# B&R Automation Studio project AS_Target_Simulink_Test
Automation Studio 4.5.2.102; This project is for testing the As Target for simulink (Third-Party Program).

## Configuration Config1

CPU PC_any, AutomationRuntime D4.52, Build 4.1.2, Vc V4.52.0

### Hardware
```
PC : PC_any v1.1.0.0 (OrderNumber=PC)
  ConfigurationID = AS_Target_Simulink_Test_Config1
  SystemTick = 1000
  Cyclic1Duration = 10000
  Cyclic1Tolerance = 10000
  ActivateOpcUa = 1
  OpcUaPort = 4841
  OpcUa_AuthenticationSecurityPolicy_EnableNone = 1
  OpcUaInformationModels_PV_Version = 1
```

## Logical view

Binary libraries used (declarations not repeated): operator, runtime, astime, AsIecCon, brsystem, sys_lib, AsArLog, AsTCP

### Global.typ - Global data types
```iecst
TYPE
	myOutputType : 	STRUCT
		out_Real : REAL;
		out_Int : ARRAY[0..2]OF INT;
		out_Bool : BOOL;
	END_STRUCT;
	myInputType : 	STRUCT
		in_Real : REAL;
		in_Int : ARRAY[0..2]OF INT;
		New_Member : BOOL;
	END_STRUCT;
END_TYPE
```

### Global.var - Global variables
```iecst
VAR
	start : BOOL := FALSE;
	ref : LREAL := 0; (*Reference input*)
	reset : BOOL := FALSE;
	x : ARRAY[0..3] OF LREAL := [4(0)]; (*Inverted pendulum state x*)
	y : ARRAY[0..1] OF LREAL := [2(0)]; (*Inverted pendulum output y*)
	F : LREAL := 0; (*Car force*)
END_VAR
```

### Package Logical/Libraries - Global libraries

### Library Logical/Libraries/pctr_fun (ANSIC, version 1.00.0)

#### lib_properties.txt
```
For manual assignment to hardware configuration please
add the following additional include directories:

\Logical\MATLAB_includes\R2019b\

And the following additional build options:

-lm -D MODEL=pend_ctrl_fun -D NUMST=1 -D NCSTATES=0 -D HAVESTDIO -D MODEL_HAS_DYNAMICALLY_LOADED_SFCNS=0 -D CLASSIC_INTERFACE=0 -D ALLOCATIONFCN=0 -D TID01EQ=0 -D TERMFCN=1 -D ONESTEPFCN=1 -D MAT_FILE=0 -D MULTI_INSTANCE_CODE=1 -D INTEGER_CODE=0 -D MT=0
```

#### pctrFub.c
```c
/********************************************************************
 * COPYRIGHT -- Bernecker + Rainer Industrie-Elektronik Ges.m.b.H.
 ********************************************************************
 * Program: pend_ctrl_fun
 * File: pctrFub.c
 * Author: Bernecker + Rainer Industrie Elektronik Ges.m.b.H.
 * Created: Wed Mar 17 14:21:47 2010
 ********************************************************************
 * Implementation of program pend_ctrl_fun
 ********************************************************************
 * Generated with B&R Automation Studio Target for Simulink  V6.1.0
 * (ERT based)
 ********************************************************************/

#include <bur/plctypes.h>
#include "pend_ctrl_fun.h"
#include "rtwtypes.h"

/* Defines */
#define SS_TERMINATE 4
#define SS_OUTPUT 3
#define SS_INITIALIZE 2

/*  Data Types */

/**************************** GLOBAL DATA *************************************/
/*  Definitions */

/*  Declarations  */

/***************************** FILE SCOPE DATA ********************************/

/*************************** FUNCTIONS ****************************************/
#ifdef __cplusplus

unsigned long bur_heap_size = 6553500;

#endif

/*LEGACYMODE_VARIABLES*/
void pctrFub(struct pctrFub* inst)
{
  tag_RTM_pend_ctrl_fun* const pend_ctrl_fun_M = &(inst)->bur_pend_ctrl_fun;
	inst->bur_pend_ctrl_fun.blockIO = &(inst)->bur_BlockIO_pend_ctrl_fun;
	inst->bur_pend_ctrl_fun.dwork = &(inst)->bur_D_Work_pend_ctrl_fun;

  switch (inst->ssMethodType)
  {
   case SS_INITIALIZE:
    /* call model initialize function */
    pend_ctrl_fun_initialize(pend_ctrl_fun_M, inst);
    break;

   case SS_OUTPUT:
    /* call model step function */
    pend_ctrl_fun_step(pend_ctrl_fun_M, inst);

    break;

   case SS_TERMINATE:
    /* call model terminate function */
    pend_ctrl_fun_terminate(pend_ctrl_fun_M, inst);
    break;
  }
}

/*****************************************************************************
   Function block sample time: 0.01s
 *****************************************************************************/

/*****************************************************************************
   B&R Automation Studio Target for Simulink Version: A6.1.0 (06-Nov-2019)
 *****************************************************************************/

/*======================== TOOL VERSION INFORMATION ==========================*
 * MATLAB 9.7 (R2019b)18-Jul-2019                                             *
 * Simulink 10.0 (R2019b)18-Jul-2019                                          *
 * Simulink Coder 9.2 (R2019b)18-Jul-2019                                     *
 * Embedded Coder 7.3 (R2019b)18-Jul-2019                                     *
 * Stateflow 10.1 (R2019b)18-Jul-2019                                         *
 * Fixed-Point Designer 6.4 (R2019b)18-Jul-2019                               *
 *============================================================================*/

/*======================= LICENSE IN USE INFORMATION =========================*
 * control_toolbox                                                            *
 * image_toolbox                                                              *
 * matlab                                                                     *
 * matlab_coder                                                               *
 * opc_toolbox                                                                *
 * real-time_workshop                                                         *
 * rtw_embedded_coder                                                         *
 * simulink                                                                   *
 *============================================================================*/
```

#### pctr_fun.fun
```iecst
FUNCTION_BLOCK pctrFub
	VAR_INPUT
		ssMethodType : SINT;
		ref : LREAL; (*Reference input*)
		x : ARRAY[0..3] OF LREAL; (*Inverted pendulum state x*)
		y : ARRAY[0..1] OF LREAL; (*Inverted pendulum output y*)
	END_VAR
	VAR_OUTPUT
		err_code : UINT; (*Controller error code*)
		F : LREAL; (*Car force*)
	END_VAR
	VAR
		bur_BlockIO_pend_ctrl_fun : BlockIO_pend_ctrl_fun;
		bur_D_Work_pend_ctrl_fun : D_Work_pend_ctrl_fun;
		bur_pend_ctrl_fun : tag_RTM_pend_ctrl_fun;
	END_VAR
END_FUNCTION_BLOCK
```

#### pctr_fun.typ
```iecst
TYPE
	BlockIO_pend_ctrl_fun :  STRUCT
		Input :  LREAL;
		Input_b :  ARRAY[0..3] OF LREAL;
		Input1 :  ARRAY[0..1] OF LREAL;
		u :  LREAL;
		err_code :  UINT;
	END_STRUCT;

	D_Work_pend_ctrl_fun :  STRUCT
		local_err_code :  UINT;
	END_STRUCT;

	tag_RTM_pend_ctrl_fun :  STRUCT
		errorStatus :  REFERENCE TO USINT;
		blockIO :  REFERENCE TO BlockIO_pend_ctrl_fun;
		dwork :  REFERENCE TO D_Work_pend_ctrl_fun;
	END_STRUCT;

	RT_MODEL_pend_ctrl_fun :tag_RTM_pend_ctrl_fun;	(*  *)

END_TYPE
```

#### pend_ctrl_fun.c
```c
/********************************************************************
 * COPYRIGHT -- Bernecker + Rainer Industrie-Elektronik Ges.m.b.H.
 ********************************************************************
 * Program: pend_ctrl_fun
 * File: pend_ctrl_fun.c
 * Author: Bernecker + Rainer Industrie Elektronik Ges.m.b.H.
 * Created: Wed Mar 17 14:21:47 2010
 ********************************************************************
 * Implementation of program pend_ctrl_fun
 ********************************************************************
 * Generated with B&R Automation Studio Target for Simulink  V6.1.0
 * (ERT based)
 ********************************************************************/

#include "pend_ctrl_fun.h"
#include "pend_ctrl_fun_private.h"

/*  Defines */

/*  Data Types */

/**************************** GLOBAL DATA *************************************/
/*  Definitions */

/*  Declarations  */

/***************************** FILE SCOPE DATA ********************************/

/*************************** FUNCTIONS ****************************************/

/* Model step function */
void pend_ctrl_fun_step(RT_MODEL_pend_ctrl_fun *const pend_ctrl_fun_M, struct pctrFub* inst)
{
  struct BlockIO_pend_ctrl_fun *pend_ctrl_fun_B = ((struct BlockIO_pend_ctrl_fun *)
    pend_ctrl_fun_M->blockIO);
  struct D_Work_pend_ctrl_fun *pend_ctrl_fun_DWork = ((struct D_Work_pend_ctrl_fun *)
    pend_ctrl_fun_M->dwork);
  real_T ref;
  uint16_T err_code;
  boolean_T varargin_1_idx_0;

  /* S-Function (bur_in): '<S1>/Input' */
  pend_ctrl_fun_B->Input = inst->ref;

  /* S-Function (bur_in): '<S4>/Input' */
  pend_ctrl_fun_B->Input_b[0] = inst->x[0];
  pend_ctrl_fun_B->Input_b[1] = inst->x[1];
  pend_ctrl_fun_B->Input_b[2] = inst->x[2];
  pend_ctrl_fun_B->Input_b[3] = inst->x[3];

  /* MATLAB Function: '<Root>/State feedback controller  with error handling' incorporates:
   *  Constant: '<Root>/ref_limit'
   *  Constant: '<Root>/u_limit'
   */
  ref = pend_ctrl_fun_B->Input;

  /* MATLAB Function 'State feedback controller  with error handling': '<S3>:1' */
  /* '<S3>:1:25' */
  err_code = pend_ctrl_fun_DWork->local_err_code;
  varargin_1_idx_0 = (fabs(pend_ctrl_fun_B->Input_b[0]) > 100.0);
  varargin_1_idx_0 = (((int32_T)varargin_1_idx_0 < (fabs
    (pend_ctrl_fun_B->Input_b[1]) > 100.0)) || varargin_1_idx_0);
  varargin_1_idx_0 = (((int32_T)varargin_1_idx_0 < (fabs
    (pend_ctrl_fun_B->Input_b[2]) > 100.0)) || varargin_1_idx_0);
  varargin_1_idx_0 = (((int32_T)varargin_1_idx_0 < (fabs
    (pend_ctrl_fun_B->Input_b[3]) > 100.0)) || varargin_1_idx_0);
  if (varargin_1_idx_0) {
    /* '<S3>:1:27' */
    /* '<S3>:1:28' */
    err_code = 50001U;

    /* '<S3>:1:29' */
    ref = 0.0;
  } else {
    if (pend_ctrl_fun_B->Input > 1.5) {
      /* '<S3>:1:31' */
      /* '<S3>:1:32' */
      err_code = 50013U;

      /* '<S3>:1:33' */
      ref = 1.5;
    } else {
      if (pend_ctrl_fun_B->Input < -1.5) {
        /* '<S3>:1:34' */
        /* '<S3>:1:35' */
        err_code = 50014U;

        /* '<S3>:1:36' */
        ref = -1.5;
      }
    }

    /* '<S3>:1:38' */
    ref = (((2987.4616903679125 * pend_ctrl_fun_B->Input_b[0] +
             3740.1178916812455 * pend_ctrl_fun_B->Input_b[1]) +
            32774.860875805127 * pend_ctrl_fun_B->Input_b[2]) +
           7399.4348019785593 * pend_ctrl_fun_B->Input_b[3]) +
      -2987.4616903679112 * ref;
    if (ref > 10000.0) {
      /* '<S3>:1:39' */
      /* '<S3>:1:40' */
      ref = 10000.0;

      /* '<S3>:1:41' */
      err_code = 50011U;
    } else {
      if (ref < -10000.0) {
        /* '<S3>:1:42' */
        /* '<S3>:1:43' */
        ref = -10000.0;

        /* '<S3>:1:44' */
        err_code = 50012U;
      }
    }
  }

  /* '<S3>:1:47' */
  pend_ctrl_fun_DWork->local_err_code = err_code;
  pend_ctrl_fun_B->u = ref;
  pend_ctrl_fun_B->err_code = err_code;

  /* End of MATLAB Function: '<Root>/State feedback controller  with error handling' */

  /* S-Function (bur_out): '<Root>/Output' */
  inst->err_code = pend_ctrl_fun_B->err_code;

  /* S-Function (bur_in): '<S4>/Input1' */
  pend_ctrl_fun_B->Input1[0] = inst->y[0];
  pend_ctrl_fun_B->Input1[1] = inst->y[1];

  /* S-Function (bur_out): '<S4>/Output' */
  inst->F = pend_ctrl_fun_B->u;
}

/* Model initialize function */
void pend_ctrl_fun_initialize(RT_MODEL_pend_ctrl_fun *const pend_ctrl_fun_M, struct pctrFub* inst)
{
  /* (no initialization code required) */
  UNUSED_PARAMETER(pend_ctrl_fun_M);
}

/* Model terminate function */
void pend_ctrl_fun_terminate(RT_MODEL_pend_ctrl_fun *const pend_ctrl_fun_M, struct pctrFub* inst)
{
  /* (no terminate code required) */
  UNUSED_PARAMETER(pend_ctrl_fun_M);
}

/*======================== TOOL VERSION INFORMATION ==========================*
 * MATLAB 9.7 (R2019b)18-Jul-2019                                             *
 * Simulink 10.0 (R2019b)18-Jul-2019                                          *
 * Simulink Coder 9.2 (R2019b)18-Jul-2019                                     *
 * Embedded Coder 7.3 (R2019b)18-Jul-2019                                     *
 * Stateflow 10.1 (R2019b)18-Jul-2019                                         *
 * Fixed-Point Designer 6.4 (R2019b)18-Jul-2019                               *
 *============================================================================*/

/*======================= LICENSE IN USE INFORMATION =========================*
 * control_toolbox                                                            *
 * image_toolbox                                                              *
 * matlab                                                                     *
 * matlab_coder                                                               *
 * opc_toolbox                                                                *
 * real-time_workshop                                                         *
 * rtw_embedded_coder                                                         *
 * simulink                                                                   *
 *============================================================================*/
```

#### pend_ctrl_fun.h
```c
/********************************************************************
 * COPYRIGHT -- Bernecker + Rainer Industrie-Elektronik Ges.m.b.H.
 ********************************************************************
 * Program: pend_ctrl_fun
 * File: pend_ctrl_fun.h
 * Author: Bernecker + Rainer Industrie Elektronik Ges.m.b.H.
 * Created: Wed Mar 17 14:21:47 2010
 ********************************************************************
 * Header for program pend_ctrl_fun
 ********************************************************************
 * Generated with B&R Automation Studio Target for Simulink  V6.1.0
 * (ERT based)
 ********************************************************************/

#ifndef RTW_HEADER_pend_ctrl_fun_h_
#define RTW_HEADER_pend_ctrl_fun_h_
#include <math.h>
#ifndef pend_ctrl_fun_COMMON_INCLUDES_
# define pend_ctrl_fun_COMMON_INCLUDES_
#include "rtwtypes.h"
#endif                                 /* pend_ctrl_fun_COMMON_INCLUDES_ */

#include "pend_ctrl_fun_types.h"
#include "pctr_fun.h"
/* Beginning of Dynamic TypeDefs: */
/* End of Dynamic TypeDefs: */
#ifndef MIN
#define MIN(a,b)	((a) < (b) ? (a) : (b))
#endif

#ifndef MAX
#define MAX(a,b)	((a) > (b) ? (a) : (b))
#endif

#ifndef AST_ROUND
#define AST_ROUND(x) ((x)>=0?(long long)((x)+0.5):(long long)((x)-0.5))
#endif

#include "rt_defines.h"

/* Macros for accessing real-time model data structure */
#ifndef rtmGetBlockIO
# define rtmGetBlockIO(rtm)            ((rtm)->blockIO)
#endif

#ifndef rtmSetBlockIO
# define rtmSetBlockIO(rtm, val)       ((rtm)->blockIO = (val))
#endif

#ifndef rtmGetRootDWork
# define rtmGetRootDWork(rtm)          ((rtm)->dwork)
#endif

#ifndef rtmSetRootDWork
# define rtmSetRootDWork(rtm, val)     ((rtm)->dwork = (val))
#endif

#ifndef rtmGetErrorStatus
# define rtmGetErrorStatus(rtm)        ((rtm)->errorStatus)
#endif

#ifndef rtmSetErrorStatus
# define rtmSetErrorStatus(rtm, val)   ((rtm)->errorStatus = (val))
#endif

#ifndef MIN
#define MIN(a,b)                       ((a) < (b) ? (a) : (b))
#endif

#ifndef MAX
#define MAX(a,b)                       ((a) > (b) ? (a) : (b))
#endif

/* Block signals (default storage) */

/* Block states (default storage) for system '<Root>' */

/* Real-time Model Data Structure */

/* Model entry point functions */
extern void pend_ctrl_fun_initialize(RT_MODEL_pend_ctrl_fun *const
  pend_ctrl_fun_M, struct pctrFub* inst);
extern void pend_ctrl_fun_step(RT_MODEL_pend_ctrl_fun *const pend_ctrl_fun_M, struct pctrFub* inst);
extern void pend_ctrl_fun_terminate(RT_MODEL_pend_ctrl_fun *const
  pend_ctrl_fun_M, struct pctrFub* inst);

/*-
 * The generated code includes comments that allow you to trace directly
 * back to the appropriate location in the model.  The basic format
 * is <system>/block_name, where system is the system number (uniquely
 * assigned by Simulink) and block_name is the name of the block.
 *
 * Use the MATLAB hilite_system command to trace the generated code back
 * to the model.  For example,
 *
 * hilite_system('<S3>')    - opens system 3
 * hilite_system('<S3>/Kp') - opens and selects block Kp which resides in S3
 *
 * Here is the system hierarchy for this model
 *
 * '<Root>' : 'pend_ctrl_fun'
 * '<S1>'   : 'pend_ctrl_fun/B&R reference input'
 * '<S2>'   : 'pend_ctrl_fun/Inverted Pendulum (Simulation // IOs)'
 * '<S3>'   : 'pend_ctrl_fun/State feedback controller  with error handling'
 * '<S4>'   : 'pend_ctrl_fun/Inverted Pendulum (Simulation // IOs)/inverted_pendulum_IOs'
 */
#endif                                 /* RTW_HEADER_pend_ctrl_fun_h_ */
```

#### pend_ctrl_fun_private.h
```c
/********************************************************************
 * COPYRIGHT -- Bernecker + Rainer Industrie-Elektronik Ges.m.b.H.
 ********************************************************************
 * Program: pend_ctrl_fun
 * File: pend_ctrl_fun_private.h
 * Author: Bernecker + Rainer Industrie Elektronik Ges.m.b.H.
 * Created: Wed Mar 17 14:21:47 2010
 ********************************************************************
 * Header for program pend_ctrl_fun
 ********************************************************************
 * Generated with B&R Automation Studio Target for Simulink  V6.1.0
 * (ERT based)
 ********************************************************************/

#ifndef RTW_HEADER_pend_ctrl_fun_private_h_
#define RTW_HEADER_pend_ctrl_fun_private_h_
#include "rtwtypes.h"
#include <bur/plctypes.h>
#ifndef MIN
#define MIN(a,b)                       ((a) < (b) ? (a) : (b))
#endif

#ifndef MAX
#define MAX(a,b)                       ((a) > (b) ? (a) : (b))
#endif
#endif                                 /* RTW_HEADER_pend_ctrl_fun_private_h_ */
```

#### pend_ctrl_fun_types.h
```c
/********************************************************************
 * COPYRIGHT -- Bernecker + Rainer Industrie-Elektronik Ges.m.b.H.
 ********************************************************************
 * Program: pend_ctrl_fun
 * File: pend_ctrl_fun_types.h
 * Author: Bernecker + Rainer Industrie Elektronik Ges.m.b.H.
 * Created: Wed Mar 17 14:21:47 2010
 ********************************************************************
 * Header for program pend_ctrl_fun
 ********************************************************************
 * Generated with B&R Automation Studio Target for Simulink  V6.1.0
 * (ERT based)
 ********************************************************************/

#ifndef RTW_HEADER_pend_ctrl_fun_types_h_
#define RTW_HEADER_pend_ctrl_fun_types_h_
#ifndef MIN
#define MIN(a,b)                       ((a) < (b) ? (a) : (b))
#endif

#ifndef MAX
#define MAX(a,b)                       ((a) > (b) ? (a) : (b))
#endif

/* Forward declaration for rtModel */

#endif                                 /* RTW_HEADER_pend_ctrl_fun_types_h_ */
```

#### rt_defines.h
```c
/********************************************************************
 * COPYRIGHT -- Bernecker + Rainer Industrie-Elektronik Ges.m.b.H.
 ********************************************************************
 * Program: pend_ctrl_fun
 * File: rt_defines.h
 * Author: Bernecker + Rainer Industrie Elektronik Ges.m.b.H.
 * Created: Wed Mar 17 14:21:47 2010
 ********************************************************************
 * Header for program pend_ctrl_fun
 ********************************************************************
 * Generated with B&R Automation Studio Target for Simulink  V6.1.0
 * (ERT based)
 ********************************************************************/

#ifndef RTW_HEADER_rt_defines_h_
#define RTW_HEADER_rt_defines_h_
#ifndef MIN
#define MIN(a,b)                       ((a) < (b) ? (a) : (b))
#endif

#ifndef MAX
#define MAX(a,b)                       ((a) > (b) ? (a) : (b))
#endif

/*===========*
 * Constants *
 *===========*/
#define RT_PI                          3.14159265358979323846
#define RT_PIF                         3.1415927F
#define RT_LN_10                       2.30258509299404568402
#define RT_LN_10F                      2.3025851F
#define RT_LOG10E                      0.43429448190325182765
#define RT_LOG10EF                     0.43429449F
#define RT_E                           2.7182818284590452354
#define RT_EF                          2.7182817F

/*
 * UNUSED_PARAMETER(x)
 *   Used to specify that a function parameter (argument) is required but not
 *   accessed by the function body.
 */
#ifndef UNUSED_PARAMETER
# if defined(__LCC__)
#   define UNUSED_PARAMETER(x)                                   /* do nothing */
# else

/*
 * This is the semi-ANSI standard way of indicating that an
 * unused function parameter is required.
 */
#   define UNUSED_PARAMETER(x)         (void) (x)
# endif
#endif
#endif                                 /* RTW_HEADER_rt_defines_h_ */
```

#### rtwtypes.h
```c
/********************************************************************
 * COPYRIGHT -- Bernecker + Rainer Industrie-Elektronik Ges.m.b.H.
 ********************************************************************
 * Program: pend_ctrl_fun
 * File: rtwtypes.h
 * Author: Bernecker + Rainer Industrie Elektronik Ges.m.b.H.
 * Created: Wed Mar 17 14:21:47 2010
 ********************************************************************
 * Header for program pend_ctrl_fun
 ********************************************************************
 * Generated with B&R Automation Studio Target for Simulink  V6.1.0
 * (ERT based)
 ********************************************************************/

#ifndef RTWTYPES_H
#define RTWTYPES_H

/* Logical type definitions */
#if (!defined(__cplusplus))
#  ifndef false
#   define false                       (0U)
#  endif

#  ifndef true
#   define true                        (1U)
#  endif
#endif

/*=======================================================================*
 * Target hardware information
 *   Device type: Intel->x86/Pentium
 *   Number of bits:     char:   8    short:   16    long:  32
 *                       long:  32
 *                       native word size:  32
 *   Byte ordering: LittleEndian
 *   Signed integer division rounds to: Zero
 *   Shift right on a signed integer as arithmetic shift: on
 *=======================================================================*/

/*=======================================================================*
 * Fixed width word size data types:                                     *
 *   int8_T, int16_T, int32_T     - signed 8, 16, or 32 bit integers     *
 *   uint8_T, uint16_T, uint32_T  - unsigned 8, 16, or 32 bit integers   *
 *   real32_T, real64_T           - 32 and 64 bit floating point numbers *
 *=======================================================================*/
typedef signed char int8_T;
typedef unsigned char uint8_T;
typedef short int16_T;
typedef unsigned short uint16_T;
typedef long int32_T;
typedef unsigned long uint32_T;
typedef float real32_T;
typedef double real64_T;

/*===========================================================================*
 * Generic type definitions: boolean_T, char_T, byte_T, int_T, uint_T,       *
 *                           real_T, time_T, ulong_T.                        *
 *===========================================================================*/
typedef double real_T;
typedef double time_T;
typedef unsigned char boolean_T;
typedef long int_T;
typedef unsigned long uint_T;
typedef unsigned long ulong_T;
typedef char char_T;
typedef unsigned char uchar_T;
typedef char_T byte_T;

/*=======================================================================*
 * Min and Max:                                                          *
 *   int8_T, int16_T, int32_T     - signed 8, 16, or 32 bit integers     *
 *   uint8_T, uint16_T, uint32_T  - unsigned 8, 16, or 32 bit integers   *
 *=======================================================================*/
#define MAX_int8_T                     ((int8_T)(127))
#define MIN_int8_T                     ((int8_T)(-128))
#define MAX_uint8_T                    ((uint8_T)(255U))
#define MAX_int16_T                    ((int16_T)(32767))
#define MIN_int16_T                    ((int16_T)(-32768))
#define MAX_uint16_T                   ((uint16_T)(65535U))
#define MAX_int32_T                    ((int32_T)(2147483647))
#define MIN_int32_T                    ((int32_T)(-2147483647-1))
#define MAX_uint32_T                   ((uint32_T)(0xFFFFFFFFU))

/* Block D-Work pointer type */
typedef void * pointer_T;

#endif                                 /* RTWTYPES_H */

#ifndef MIN
#define MIN(a,b)                       ((a) < (b) ? (a) : (b))
#endif

#ifndef MAX
#define MAX(a,b)                       ((a) > (b) ? (a) : (b))
#endif
```

### Package Logical/MATLAB_includes - Default includes for B&R Automation Studio Target for Simulink

### MatlabDataArray.hpp
```cpp
/* Copyright 2016-2017 The MathWorks, Inc. */

#ifndef MATLAB_DATA_ARRAY_HPP
#define MATLAB_DATA_ARRAY_HPP

#include "MatlabDataArray/Exception.hpp"
#include "MatlabDataArray/matlab_data_array_defs.hpp"
#include "MatlabDataArray/matlab_extdata_defs.hpp"
#include "MatlabDataArray/ArrayDimensions.hpp"
#include "MatlabDataArray/ArrayType.hpp"
#include "MatlabDataArray/GetReturnType.hpp"
#include "MatlabDataArray/Range.hpp"
#include "MatlabDataArray/String.hpp"
#include "MatlabDataArray/Enumeration.hpp"
#include "MatlabDataArray/Struct.hpp"
#include "MatlabDataArray/Reference.hpp"
#include "MatlabDataArray/ArrayElementRef.hpp"
#include "MatlabDataArray/ArrayElementTypedRef.hpp"
#include "MatlabDataArray/ArrayReferenceExt.hpp"
#include "MatlabDataArray/TypedArrayRef.hpp"
#include "MatlabDataArray/ArrayFactory.hpp"
#include "MatlabDataArray/TypedIterator.hpp"
#include "MatlabDataArray/ForwardIterator.hpp"
#include "MatlabDataArray/TypedArray.hpp"
#include "MatlabDataArray/StructRef.hpp"
#include "MatlabDataArray/SparseArray.hpp"
#include "MatlabDataArray/SparseArrayRef.hpp"
#include "MatlabDataArray/EnumArray.hpp"
#include "MatlabDataArray/MatlabFieldIdentifier.hpp"
#include "MatlabDataArray/StructArray.hpp"
#include "MatlabDataArray/CharArray.hpp"
#include "MatlabDataArray/ArrayVisitors.hpp"
#include "MatlabDataArray/Optional.hpp"

#endif
```

### covrt.h
```c
/*
 * PUBLISHED header for covrt, the runtime library for Code Coverage
 *
 * Copyright 1984-2013 The MathWorks, Inc.
 *
 */

#ifndef covrt_h
#define covrt_h

#if defined(_MSC_VER)
# pragma once
#endif
#if defined(__GNUC__) && (__GNUC__ > 3 || (__GNUC__ == 3 && __GNUC_MINOR__ > 3))
# pragma once
#endif

/*
 * Only define EXTERN_C if it hasn't been defined already. This allows
 * individual modules to have more control over managing their exports.
 */
#ifndef EXTERN_C

#ifdef __cplusplus
#define EXTERN_C extern "C"
#else
#define EXTERN_C extern
#endif

#endif

#ifndef LIBCOVRT_API
#define LIBCOVRT_API
#endif

#include <setjmp.h>
#include <stdio.h>
#include "matrix.h"

/*
 * MATLAB INTERNAL USE ONLY :: Instance specific runtime data.
 */
typedef struct covrtInstanceData covrtInstanceData;

/*
 * MATLAB INTERNAL USE ONLY :: Instance type
 */
typedef struct covrtInstance {
    covrtInstanceData* data;
} covrtInstance;

/* one instance per mex */
extern covrtInstance gCoverageLoggingInstance;

typedef struct CovrtStateflowData CovrtStateflowData;

typedef struct CovrtStateflowInstance {
	CovrtStateflowData*  data;
	double instanceHandle;
} CovrtStateflowInstance;

/*
 * MATLAB INTERNAL USE ONLY :: Enable/Disable Coverage Logging during mex execution
 */
EXTERN_C LIBCOVRT_API void covrtEnableCoverageLogging( bool enable );

/*
 * MATLAB INTERNAL USE ONLY :: Enabled/Disable use of cv.mex
 */
EXTERN_C LIBCOVRT_API void covrtUseCV(bool useCV);

/*
 * MATLAB INTERNAL USE ONLY :: reset flag
 */
EXTERN_C LIBCOVRT_API void covrtResetUpdateFlag();

/*
 * MATLAB INTERNAL USE ONLY :: Allocate instance data
 */
EXTERN_C LIBCOVRT_API void covrtAllocateInstanceData( covrtInstance* instance );

/*
 * MATLAB INTERNAL USE ONLY :: Free instance data
 */
EXTERN_C LIBCOVRT_API void covrtFreeInstanceData( covrtInstance* instance );

/*
 * MATLAB INTERNAL USE ONLY :: Free instance data
 */
EXTERN_C LIBCOVRT_API mxArray* covrtSerializeInstanceData( covrtInstance* instance );

/*
 * MATLAB INTERNAL USE ONLY :: Coverage engine script initalization callback
 */
EXTERN_C LIBCOVRT_API void covrtScriptStart(covrtInstance* instance,
                                            unsigned int cvId);

/*
 * MATLAB INTERNAL USE ONLY :: Initialize Script
 */
EXTERN_C LIBCOVRT_API void covrtScriptInit( covrtInstance* instance,
                                            const char* path,
                                            unsigned int cvId,
                                            unsigned int fcnCnt,
                                            unsigned int basicBlockCnt,
                                            unsigned int ifCnt,
                                            unsigned int testobjectiveCnt,
	                                    unsigned int saturationCnt,
                                            unsigned int switchCnt,
                                            unsigned int forCnt,
                                            unsigned int whileCnt,
                                            unsigned int condCnt,
                                            unsigned int mcdcCnt);

/*
 * MATLAB INTERNAL USE ONLY :: Initialize Function
 */
EXTERN_C LIBCOVRT_API void covrtFcnInit( covrtInstance* instance,
                                         unsigned int cvId,
                                         unsigned int fcnIdx,
                                         const char *name,
                                         int charStart,
                                         int charExprEnd,
                                         int charEnd);

/*
 * MATLAB INTERNAL USE ONLY :: Initialize Basic Block
 */
EXTERN_C LIBCOVRT_API void covrtBasicBlockInit( covrtInstance* instance,
                                         unsigned int cvId,
                                         unsigned int fcnIdx,
                                         int charStart,
                                         int charExprEnd,
                                         int charEnd);

/*
 * MATLAB INTERNAL USE ONLY :: Initialize If
 */
EXTERN_C LIBCOVRT_API void covrtIfInit( covrtInstance* instance,
                                        unsigned int cvId,
                                        unsigned int ifIdx,
                                        int charStart,
                                        int charExprEnd,
                                        int charElseStart,
                                        int charEnd);

/*
 * MATLAB INTERNAL USE ONLY :: Initialize Mcdc
 */
EXTERN_C LIBCOVRT_API void covrtMcdcInit( covrtInstance* instance,
                                          unsigned int cvId,
                                          unsigned int mcdcIdx,
                                          int charStart,
                                          int charEnd,
                                          int condCnt,
                                          int firstCondIdx,
                                          int* condStart,
                                          int* condEnd,
                                          int postFixLength,
                                          int* postFixExprs);

/*
 * MATLAB INTERNAL USE ONLY :: Initialize Switch
 */
EXTERN_C LIBCOVRT_API void covrtSwitchInit( covrtInstance* instance,
                                            unsigned int cvId,
                                            unsigned int switchIdx,
                                            int charStart,
                                            int charExprEnd,
                                            int charEnd,
                                            unsigned int caseCnt,
                                            int *caseStart,
                                            int *caseExprEnd);

/*
 * MATLAB INTERNAL USE ONLY :: Initialize For
 */
EXTERN_C LIBCOVRT_API void covrtForInit( covrtInstance* instance,
                                         unsigned int cvId,
                                         unsigned int forIdx,
                                         int charStart,
                                         int charExprEnd,
                                         int charEnd);

/*
 * MATLAB INTERNAL USE ONLY :: Initialize While
 */
EXTERN_C LIBCOVRT_API void covrtWhileInit( covrtInstance* instance,
                                           unsigned int cvId,
                                           unsigned int whileIdx,
                                           int charStart,
                                           int charExprEnd,
                                           int charEnd);

/*
 * MATLAB INTERNAL USE ONLY :: Initialize MCDC
 */
EXTERN_C LIBCOVRT_API void covrtMCDCInit( covrtInstance* instance,
                                          unsigned int cvId,
                                          unsigned int mcdcIdx,
                                          int charStart,
                                          int charEnd,
                                          unsigned int condCnt,
                                          unsigned int firstCondIdx,
                                          int *condStart,
                                          int *condEnd,
                                          unsigned int pfxLength,
                                          int *pfixExpr);

/*
 * MATLAB INTERNAL USE ONLY :: Log Function
 */
EXTERN_C LIBCOVRT_API void covrtLogFcn(covrtInstance* instance,
                                       uint32_T covId,
                                       uint32_T fcnId);

/*
 * MATLAB INTERNAL USE ONLY :: Log Basic Block
 */
EXTERN_C LIBCOVRT_API void covrtLogBasicBlock(covrtInstance* instance,
                                       uint32_T covId,
                                       uint32_T basicBlockId);

/*
 * MATLAB INTERNAL USE ONLY :: Log If
 */
EXTERN_C LIBCOVRT_API int32_T covrtLogIf(covrtInstance* instance,
                                         uint32_T covId,
                                         uint32_T fcnId,
                                         int32_T ifId,
                                         int32_T condition);

/*
 * MATLAB INTERNAL USE ONLY :: Log Cond
 */
EXTERN_C LIBCOVRT_API int32_T covrtLogCond(covrtInstance* instance,
                                            uint32_T covId,
                                            uint32_T fcnId,
                                            int32_T condId,
                                            int32_T condition);

/*
 * MATLAB INTERNAL USE ONLY :: Log If
 */
EXTERN_C LIBCOVRT_API void covrtLogFor(covrtInstance* instance,
                                        uint32_T covId,
                                        uint32_T fcnId,
                                        int32_T forId,
                                        int32_T entryOrExit);

/*
 * MATLAB INTERNAL USE ONLY :: Log While
 */
EXTERN_C LIBCOVRT_API int32_T covrtLogWhile(covrtInstance* instance,
                                            uint32_T covId,
                                            uint32_T fcnId,
                                            int32_T whileId,
                                            int32_T condition);

/*
 * MATLAB INTERNAL USE ONLY :: Log Switch
 */
EXTERN_C LIBCOVRT_API void covrtLogSwitch(covrtInstance* instance,
                                            uint32_T covId,
                                            uint32_T fcnId,
                                            int32_T switchId,
                                            int32_T caseId);

/*
 * MATLAB INTERNAL USE ONLY :: Log If
 */
EXTERN_C LIBCOVRT_API int32_T covrtLogMcdc(covrtInstance* instance,
                                            uint32_T covId,
                                            uint32_T fcnId,
                                            int32_T mcdcId,
                                            int32_T condition);

/*
 * MATLAB INTERNAL USE ONLY :: Log decision in block
 */
EXTERN_C LIBCOVRT_API int32_T covrtLogBlockDec(covrtInstance* instance,
                                            uint32_T covId,
                                            int32_T decId,
                                            int32_T eleIdx,
                                            int32_T decVal);

/* stateflow */

EXTERN_C LIBCOVRT_API
void covrtCreateStateflowInstance(CovrtStateflowInstance* instance,
	unsigned int stateCount,
	unsigned int eventCount,
	unsigned int transCount,
	unsigned int dataCount);

EXTERN_C LIBCOVRT_API
void covrtSetInstanceCvIds(
	unsigned int cvChartId,
	double* cvStateIds,
	size_t stateCnt,
	double* cvTransIds,
	size_t transCnt);

EXTERN_C LIBCOVRT_API
void covrtDeleteStateflowInstance(CovrtStateflowInstance* instance);

EXTERN_C LIBCOVRT_API void covrtRelationalopInitFcn(
	CovrtStateflowInstance* instance,
	unsigned int transitionNumber,
	unsigned int relopCnt,
	int* txtStartIdx,
	int* txtEndIdx,
	int* relationalEps,
	int* relationalOp);

EXTERN_C LIBCOVRT_API void covrtSaturationInitFcn(
	CovrtStateflowInstance* instance,
	unsigned int objectType,
	unsigned int transitionNumber,
	unsigned int satCnt,
	unsigned int* txtStartIdx,
	unsigned int* txtEndIdx);

EXTERN_C LIBCOVRT_API void covrtTransInitFcn(CovrtStateflowInstance* instance,
	unsigned int transitionNumber,
	int predicateCnt,
	unsigned int* txtStartIdx,
	unsigned int* txtEndIdx,
	unsigned int postFixPredicateTreeCount,
	int* postFixPredicateTree);

EXTERN_C LIBCOVRT_API void covrtStateInitFcn(CovrtStateflowInstance* instance,
	unsigned int stateNumber,
	unsigned int numChild,
	bool hasDuringSwitch,
	bool hasExitSwitch,
	bool hasHistSwitch,
	unsigned int onDecCnt,
	unsigned int* decStartInd,
	unsigned int* decEndInd);

EXTERN_C LIBCOVRT_API void covrtChartInitFcn(CovrtStateflowInstance* instance,
	unsigned int numChild,
	bool hasDuringSwitch,
	bool hasExitSwitch,
	bool hasHistSwitch);

EXTERN_C LIBCOVRT_API unsigned int covrtRelationalopUpdateFcn(CovrtStateflowInstance* instance,
	unsigned int objectType,
	unsigned int objectNumber,
	unsigned int objectIndex,
	double lhsVal,
	double rhsVal,
	int relationalopEps,
	unsigned int op,
	int retValue);

EXTERN_C LIBCOVRT_API unsigned int covrtSaturationUpdateFcn(CovrtStateflowInstance* instance,
	unsigned int objectType,
	unsigned int objectNumber,
	unsigned int satIdx,
	unsigned int isNeg,
	int val);

EXTERN_C LIBCOVRT_API void covrtSaturationUpdateAccumFcn(CovrtStateflowInstance* instance,
	unsigned int objectType,
	unsigned int objectNumber,
	unsigned int satIdx,
	unsigned int accumMode);

EXTERN_C LIBCOVRT_API unsigned int covrtDecUpdateFcn(CovrtStateflowInstance* instance,
	unsigned int objectType,
	unsigned int objectNumber,
	unsigned int objectIndex,
	unsigned int retValue);

EXTERN_C LIBCOVRT_API unsigned int covrtCondUpdateFcn(CovrtStateflowInstance* instance,
	unsigned int objectType,
	unsigned int objectNumber,
	unsigned int objectIndex,
	unsigned int retValue);

EXTERN_C LIBCOVRT_API unsigned int covrtSigUpdateFcn(CovrtStateflowInstance* instance,
	unsigned int dataNumber,
	double equivValue);

#endif /* covrt_h */
```

### slexec_block_runtime_service.h
```c
#ifndef SIMSTRUCT_SLEXEC_BLOCK_RUNTIME_SERVICE_H
#define SIMSTRUCT_SLEXEC_BLOCK_RUNTIME_SERVICE_H

/**
 * @file slexec_block_runtime_service.h
 *
 * This header is the exported C interface to the simulink execution engine
 * (slexec_simbridge) that provides block runtime services. This file should be
 * included from simstruct (and no earlier) so that we have access to
 * preprocessor variables.
 *
 * Note that this header file should be placed in the simstruct folder, and its
 * implementations are in the simbridge module.
 *
 */

/* Copyright 2017 The MathWorks, Inc. */

/* Guard against early inclusions */
#ifndef _SIMSTRUCT
#error "This file should be included from simstruc.h"
#endif

#ifdef BUILDING_SLEXEC_SIMBRIDGE
 /* being included from inside slexec_simbridge module */
  #include "package.h"
  #define SLEXEC_SIMBRIDGE_PUBLISHED_C extern "C" DLL_EXPORT_SYM
#else
 /* being included from outside, such as raccel code */
  #if defined(__cplusplus)
 /* Needed for non-inlined C++ S-functions */
    #define SLEXEC_SIMBRIDGE_PUBLISHED_C extern "C"
  #else
    #define SLEXEC_SIMBRIDGE_PUBLISHED_C extern
  #endif
#endif

/* Block runtime service keys */
typedef enum {
    SLEXEC_BLK_RTS_SET_NUM_TICKS_TO_NEXT_SAMPLE_HIT_FOR_VDR,
    SLEXEC_BLK_RTS_GET_NUM_TICKS_TO_NEXT_SAMPLE_HIT_FOR_VDR
} _slexecBlkRTSType;

/* Type declarations */
typedef int_T  (*_slexecBlkRTSGateway) (SimStruct*        S,
                                        _slexecBlkRTSType type,
                                        int_T             arg1,
                                        void*             arg2);

/* Macro utilities */
#define _slexecSafelyCallBlkRTSGatewayStart(S) \
    (((S)->mdlInfo->blkRTSGateway==NULL) ? 0 : ((*(S)->mdlInfo->blkRTSGateway)
#define _slexecSafelyCallBlkRTSGatewayEnd ))

#define _slexecSetBlkRTSGateway(S,fcn)   \
    (S)->mdlInfo->blkRTSGateway = (fcn)

/* Block runtime service function */
SLEXEC_SIMBRIDGE_PUBLISHED_C int _slexecBlockRuntimeServiceGateway(SimStruct*        S,
                                                                   _slexecBlkRTSType blkRTSType,
                                                                   int               arg1,
                                                                   void*             arg2);

/* Published block runtime service macros */

/*
 * This macro is used to set the number of ticks to the next sample hit for
 * variable discrete rate in the block.
 *
 * sti is the sample time index of the variable discrete rate in the block, and
 * numTicks is the the next ticks to the next sample hit.
 *
 */
#define ssSetNumTicksToNextSampleHitForVariableDiscrete(S, sti, numTicks)                                                 \
{                                                                                                                         \
      size_t tmp = (size_t) numTicks;                                                                                     \
      _slexecSafelyCallBlkRTSGatewayStart(S)(S, SLEXEC_BLK_RTS_SET_NUM_TICKS_TO_NEXT_SAMPLE_HIT_FOR_VDR, (int) sti, &tmp) \
      _slexecSafelyCallBlkRTSGatewayEnd;                                                                                  \
}

/*
 * This macro is used to get the number of ticks to the next sample hit for
 * variable discrete rate in the block.
 *
 * sti is the sample time index of the variable discrete rate in the block.
 *
 */
#define ssGetNumTicksToNextSampleHitForVariableDiscrete(S, sti)                                                                   \
{                                                                                                                                 \
      _slexecSafelyCallBlkRTSGatewayStart(S)(S, SLEXEC_BLK_RTS_GET_NUM_TICKS_TO_NEXT_SAMPLE_HIT_FOR_VDR, (int) sti, (void*) NULL) \
      _slexecSafelyCallBlkRTSGatewayEnd;                                                                                          \
}

#endif
```

### slexec_vm_simstruct_bridge.h
```c
#ifndef SLEXEC_VM_SIMSTRUCT_BRIDGE_H
#define SLEXEC_VM_SIMSTRUCT_BRIDGE_H
/**
 * @file slexec_vm_simstruct_bridge.h
 *
 * This header is the exported C interface of the SimStruct and related
 * data structures, for use in VM applications.
 *
 */

/* Copyright 2015-2017 The MathWorks, Inc. */

#include "tmwtypes.h"

#ifdef BUILDING_SLEXEC_SIMBRIDGE
 /* being included from inside slexec_simbridge module */
  #include "package.h"
  #define SLEXEC_SIMBRIDGE_PUBLISHED_C extern "C" DLL_EXPORT_SYM
#else
 /* being included from outside, such as raccel code */
  #if defined(__cplusplus)
 /* Needed for non-inlined C++ S-functions */
    #define SLEXEC_SIMBRIDGE_PUBLISHED_C extern "C"
  #else
    #define SLEXEC_SIMBRIDGE_PUBLISHED_C extern
  #endif
#endif

SLEXEC_SIMBRIDGE_PUBLISHED_C void vm_ssCallAccelRunBlock(
    void* S, int_T sysIdx, int_T blkIdx, int_T blkFcn);
SLEXEC_SIMBRIDGE_PUBLISHED_C void vm_ssCallAccelPreBlock(
    void* S, int_T sysIdx, int_T blkIdx, int_T blkFcn);
SLEXEC_SIMBRIDGE_PUBLISHED_C void vm_ssCallAccelPostBlock(
    void* S, int_T sysIdx, int_T blkIdx, int_T blkFcn);

SLEXEC_SIMBRIDGE_PUBLISHED_C void vm_slmrAccelRunBlockSystemInitialize(
    void* S, int_T sysIdx, int_T blkIdx);
SLEXEC_SIMBRIDGE_PUBLISHED_C void vm_slmrAccelRunBlockSystemReset(
    void* S, int_T sysIdx, int_T blkIdx);
SLEXEC_SIMBRIDGE_PUBLISHED_C void vm_ssCallAccelModelBlockFcnCallInput(
    void* S, int_T sysIdx, int_T blkIdx, int_T portIdx, int_T tid, int_T blkFcn);
SLEXEC_SIMBRIDGE_PUBLISHED_C void vm_ssCallAccelCopyCacheForIIS(
    void* S, int_T sysIdx, int_T fromCache);
SLEXEC_SIMBRIDGE_PUBLISHED_C void vm_ssCallAccelSetDims(
    void* S, int_T sysIdx, int_T blkIdx, int_T outIdx, int_T ruleIdx);
SLEXEC_SIMBRIDGE_PUBLISHED_C void vm_ssSetChecksumVal(
    void *S, int_T sysIdx, int_T blkIdx);
SLEXEC_SIMBRIDGE_PUBLISHED_C void vm__ssGetBlockPath(
    void* S, int_T sysIdx, int_T blkIdx, char_T** path);

SLEXEC_SIMBRIDGE_PUBLISHED_C void* vm_ssGetRootDWork(void* S);
SLEXEC_SIMBRIDGE_PUBLISHED_C void* vm__ssGetModelBlockIO(void* S);
SLEXEC_SIMBRIDGE_PUBLISHED_C const void* vm_ssGetConstBlockIO(void* S);
SLEXEC_SIMBRIDGE_PUBLISHED_C double* vm_ssGetModelRtp(void* S);

SLEXEC_SIMBRIDGE_PUBLISHED_C void* vm_ssGetU(void* S);
SLEXEC_SIMBRIDGE_PUBLISHED_C void* vm_ssGetUByIndex(void* S, int_T index);
SLEXEC_SIMBRIDGE_PUBLISHED_C void* vm_ssGetX(void* S);
SLEXEC_SIMBRIDGE_PUBLISHED_C void* vm_ssGetdX(void* S);
SLEXEC_SIMBRIDGE_PUBLISHED_C void* vm_ssGetAbsTolVector(void* S);
SLEXEC_SIMBRIDGE_PUBLISHED_C void* vm_ssGetY(void* S);
SLEXEC_SIMBRIDGE_PUBLISHED_C void* vm_ssGetYByIndex(void* S, int_T index);

SLEXEC_SIMBRIDGE_PUBLISHED_C void vm_dworkSizeCheck(void* S, uint_T sizeofStruct);
SLEXEC_SIMBRIDGE_PUBLISHED_C void vm_blockIOSizeCheck(void* S, uint_T sizeofStruct);
SLEXEC_SIMBRIDGE_PUBLISHED_C void vm_USizeCheck(void* S, uint_T sizeofStruct);
SLEXEC_SIMBRIDGE_PUBLISHED_C void vm_YSizeCheck(void* S, uint_T sizeofStruct);
SLEXEC_SIMBRIDGE_PUBLISHED_C void vm_paramSizeCheck(void* S, uint_T sizeofStruct);

SLEXEC_SIMBRIDGE_PUBLISHED_C int_T
    vm_ssIsSampleHit(void* S, int_T sti, int_T tid);
SLEXEC_SIMBRIDGE_PUBLISHED_C int_T vm_ssIsContinuousTask(void* S, int_T tid);
SLEXEC_SIMBRIDGE_PUBLISHED_C void vm__ssSetSampleHit(void* S, int_T sti,
                                                     int_T v);
SLEXEC_SIMBRIDGE_PUBLISHED_C int vm_ssIsSpecialSampleHit(void* S, int_T my_sti,
                                                         int_T promoted_sti,
                                                         int_T tid);

SLEXEC_SIMBRIDGE_PUBLISHED_C uint32_T vm_ssGetClockTick(void* S, int_T sti);
SLEXEC_SIMBRIDGE_PUBLISHED_C uint32_T vm_ssGetClockTickH(void* S, int_T sti);

SLEXEC_SIMBRIDGE_PUBLISHED_C double* vm_ssGetSolverZcSignalVector(void* S);
SLEXEC_SIMBRIDGE_PUBLISHED_C uint8_T* vm_ssGetPrevZCSigState(void* S);

SLEXEC_SIMBRIDGE_PUBLISHED_C int_T vm_ssIsMajorTimeStep(void* S);

SLEXEC_SIMBRIDGE_PUBLISHED_C void vm_ssSetStopRequested(void* S, int_T val);

SLEXEC_SIMBRIDGE_PUBLISHED_C void vm_srClearBC(int8_T* state);
SLEXEC_SIMBRIDGE_PUBLISHED_C void  vm_srUpdateBC(int8_T* state);

SLEXEC_SIMBRIDGE_PUBLISHED_C double vm_ssGetT(void* S);
SLEXEC_SIMBRIDGE_PUBLISHED_C double vm_ssGetTaskTime(void* S, int_T sti);
SLEXEC_SIMBRIDGE_PUBLISHED_C void vm__ssSetTaskTime(void* S, int_T sti,
                                                    double time);
SLEXEC_SIMBRIDGE_PUBLISHED_C double vm_ssGetTStart(void* S);
SLEXEC_SIMBRIDGE_PUBLISHED_C double vm_ssGetTFinal(void* S);
SLEXEC_SIMBRIDGE_PUBLISHED_C double vm_ssGetStepSize(void* S);
SLEXEC_SIMBRIDGE_PUBLISHED_C double vm_ssGetTimeOfLastOutput(void* S);

SLEXEC_SIMBRIDGE_PUBLISHED_C double vm__ssGetVarNextHitTime(void* S,
                                                            int_T varId);
SLEXEC_SIMBRIDGE_PUBLISHED_C void vm__ssSetVarNextHitTime(void* S, int_T varId,
                                                          double tNextMin);
SLEXEC_SIMBRIDGE_PUBLISHED_C void vm_ssSetTimeOfNextVarHit(void* S, int_T sti,
                                                           double tNextMin);

SLEXEC_SIMBRIDGE_PUBLISHED_C uint8_T
    vm_ssGetTNextWasAdjusted(void* S, int_T varTsId);

SLEXEC_SIMBRIDGE_PUBLISHED_C uint8_T* vm_ssGetContStateDisabled(void* S);

SLEXEC_SIMBRIDGE_PUBLISHED_C uint8_T vm_ssIsFirstInitCond(void* S);

SLEXEC_SIMBRIDGE_PUBLISHED_C const char_T* vm_ssGetErrorStatus(void* S);
SLEXEC_SIMBRIDGE_PUBLISHED_C uint8_T vm_getHasError(void* S);
SLEXEC_SIMBRIDGE_PUBLISHED_C void vm_ssSetErrorStatus(void* S,
                                                      const char_T* str);
SLEXEC_SIMBRIDGE_PUBLISHED_C void vm__ssSet_slErrMsg(void* S, void* diag);
SLEXEC_SIMBRIDGE_PUBLISHED_C void vm__ssReportDiagnosticAsWarning(void* S,
                                                                  void* diag);

SLEXEC_SIMBRIDGE_PUBLISHED_C void vm_ssSetContTimeOutputInconsistentWithStateAtMajorStep(void* S);
SLEXEC_SIMBRIDGE_PUBLISHED_C void vm_ssSetBlockStateForSolverChangedAtMajorStep(void* S);

SLEXEC_SIMBRIDGE_PUBLISHED_C void vm_ReadLocalDSMNoIdx(void* S, int_T dsmIdx,
                                                       const char_T* blockPath,
                                                       int_T idxWidth);
SLEXEC_SIMBRIDGE_PUBLISHED_C void vm_ReadLocalDSMIntIdx(void* S, int_T dsmIdx,
                                                        const char_T* blockPath,
                                                        int_T idx,
                                                        int_T idxWidth);
SLEXEC_SIMBRIDGE_PUBLISHED_C void vm_WriteLocalDSMNoIdx(void* S, int_T dsmIdx,
                                                        const char_T* blockPath,
                                                        int_T idxWidth);
SLEXEC_SIMBRIDGE_PUBLISHED_C void vm_WriteLocalDSMIntIdx(
    void* S, int_T dsmIdx, const char_T* blockPath, int_T idx, int_T idxWidth);
SLEXEC_SIMBRIDGE_PUBLISHED_C void vm_ReadGlobalDSMNoIdx(void* S, int_T dsmIdx,
                                                        const char_T* blockPath,
                                                        int_T idxWidth);
SLEXEC_SIMBRIDGE_PUBLISHED_C void vm_ReadGlobalDSMIntIdx(
    void* S, int_T dsmIdx, const char_T* blockPath, int_T idx, int_T idxWidth);
SLEXEC_SIMBRIDGE_PUBLISHED_C void vm_WriteGlobalDSMNoIdx(
    void* S, int_T dsmIdx, const char_T* blockPath, int_T idxWidth);
SLEXEC_SIMBRIDGE_PUBLISHED_C void vm_WriteGlobalDSMIntIdx(
    void* S, int_T dsmIdx, const char_T* blockPath, int_T idx, int_T idxWidth);

SLEXEC_SIMBRIDGE_PUBLISHED_C void vm__ssIsPositiveDataValue(void* S, void* data,
                                                            int_T dtId,
                                                            int8_T* result);

SLEXEC_SIMBRIDGE_PUBLISHED_C void vm__ssSignDataValue(void* S, void* data,
                                                      int_T dtId,
                                                      int8_T* result);

SLEXEC_SIMBRIDGE_PUBLISHED_C uint8_T vm_ssIsSolverComputingJacobian(void* S);
SLEXEC_SIMBRIDGE_PUBLISHED_C uint8_T vm_ssIsSolverRequestingReset(void* S);
SLEXEC_SIMBRIDGE_PUBLISHED_C uint8_T vm_ssIsSolverCheckingCIC(void* S);

SLEXEC_SIMBRIDGE_PUBLISHED_C void vm_ssDummy();

SLEXEC_SIMBRIDGE_PUBLISHED_C uint8_T vm_ssGetEvaluatingF0ForJacobian(void* S);

SLEXEC_SIMBRIDGE_PUBLISHED_C void vm_ssSetNumTicksToNextSampleHitForVariableDiscrete(void* S,
                                                                                     int_T stIdx,
                                                                                     int8_T* numTicks);
#endif
```

### slsv_diagnostic_codegen_c_api.h
```c
/* Copyright 2010-2012 The MathWorks, Inc. */

#ifndef slsv_diagnostic_codegen_c_api_h
#define slsv_diagnostic_codegen_c_api_h

#include "tmwtypes.h"

#ifdef BUILDING_LIBMWSL_SERVICES
 /* being included from inside sl_services module */
  #include "package.h"
  #define SL_SERVICES_PUBLISHED_C extern "C" DLL_EXPORT_SYM
#else
 /* being included from outside, such as raccel code */
  #if defined(__cplusplus)
 /* Needed for non-inlined C++ S-functions */
    #define SL_SERVICES_PUBLISHED_C extern "C"
  #else
    #define SL_SERVICES_PUBLISHED_C extern
  #endif
#endif

/* for valist_CreateDiagnosticAsVoidPtr */
#if defined(__cplusplus)
  #include <cstdarg>
#else
  #include <stdarg.h>
#endif

#include "slsv_diagnostic_logger_type.h"

#define CODEGEN_SUPPORT_ARG_END_LIST             (int)0
#define CODEGEN_SUPPORT_ARG_INTEGER_TYPE (int)1
#define CODEGEN_SUPPORT_ARG_REAL_TYPE (int)2
#define CODEGEN_SUPPORT_ARG_STRING_TYPE (int)3
#define CODEGEN_SUPPORT_ARG_ENCODED_STRING_TYPE (int)4
#define CODEGEN_SUPPORT_ARG_ESCAPED_STRING_TYPE (int)5

#define CODEGEN_SUPPORT_DIAGNOSTIC_INFO (int)0
#define CODEGEN_SUPPORT_DIAGNOSTIC_WARNING (int)1
#define CODEGEN_SUPPORT_DIAGNOSTIC_ERROR (int)2

SL_SERVICES_PUBLISHED_C char* CreateDiagnosticXMLSnippet(const char* id,
                                                         int nargs, ...);

SL_SERVICES_PUBLISHED_C void* CreateDiagnosticAsVoidPtr(const char* id,
                                                        int nargs, ...);

SL_SERVICES_PUBLISHED_C void* valist_CreateDiagnosticAsVoidPtr(const char* id,
                                                               int nargs,
                                                               va_list args);

/* UTF8 path */
SL_SERVICES_PUBLISHED_C void dl_set_home(const char *path);

SL_SERVICES_PUBLISHED_C dl_logger_sid_t dl_init(size_t);
SL_SERVICES_PUBLISHED_C void dl_clear(dl_logger_sid_t);
SL_SERVICES_PUBLISHED_C void dl_destroy(dl_logger_sid_t);
SL_SERVICES_PUBLISHED_C void dl_reset(dl_logger_sid_t);

SL_SERVICES_PUBLISHED_C void dl_report(dl_logger_sid_t, int type, const char* id, ...);

/* void * from CreateDiagnosticAsVoidPtr */
SL_SERVICES_PUBLISHED_C void dl_report_from_diagnostic(dl_logger_sid_t, int type, void* diagnostic);

#endif /* slsv_diagnostic_codegen_c_api_h */
```

### tmwtypes.h
```c
/*
 * Copyright 1984-2016 The MathWorks, Inc.
 * All Rights Reserved.
 */

#if defined(_MSC_VER)
# pragma once
#endif
#if defined(__GNUC__) && (__GNUC__ > 3 || (__GNUC__ == 3 && __GNUC_MINOR__ > 3))
# pragma once
#endif

#ifndef tmwtypes_h
#define tmwtypes_h

#ifndef __TMWTYPES__
#define __TMWTYPES__
/*
 * File    : tmwtypes.h
 * Abstract:
 *      Data types for use with MATLAB/SIMULINK and the Real-Time Workshop.
 *
 *      When compiling stand-alone model code, data types can be overridden
 *      via compiler switches.
 *
 *      Define NO_FLOATS to eliminate reference to real_T, etc.
 */

#include <limits.h>

#ifdef __APPLE_CC__
#include <stdbool.h>
#endif

#define LOGICAL_IS_A_TYPE
#define SPARSE_GENERALIZATION

#ifdef NO_FLOATS
# define double double_not_allowed
# define float  float_not_allowed
#endif /*NO_FLOATS*/

#ifndef NO_FLOATS

#ifndef __MWERKS__
# ifdef __STDC__
#  include <float.h>
# else
#  define FLT_MANT_DIG 24
#  define DBL_MANT_DIG 53
# endif
#endif

#endif /*NO_FLOATS*/

/*
 *      The following data types cannot be overridden when building MEX files.
 */
#ifdef MATLAB_MEX_FILE
# undef CHARACTER_T
# undef INTEGER_T
# undef BOOLEAN_T
# undef REAL_T
# undef TIME_T
#endif

/*
 * The uchar_T, ushort_T and ulong_T types are needed for compilers which do
 * not allow defines to be specified, at the command line, with spaces in them.
 */

typedef unsigned char       uchar_T;
typedef unsigned short      ushort_T;
typedef unsigned long       ulong_T;

#if (defined(_MSC_VER) && _MSC_VER >= 1500)      \
    || defined(__x86_64__) || defined(__LP64__)  \
    || defined(__LCC64__)

typedef unsigned long long  ulonglong_T;
#endif

/*=======================================================================*
 * Fixed width word size data types:                                     *
 *   int8_T, int16_T, int32_T     - signed 8, 16, or 32 bit integers     *
 *   uint8_T, uint16_T, uint32_T  - unsigned 8, 16, or 32 bit integers   *
 *   real32_T, real64_T           - 32 and 64 bit floating point numbers *
 *=======================================================================*/

/* When used with Real Time Workshop generated code, this
 * header file can be used with a variety of compilers.
 *
 * The compiler could be for an 8 bit embedded processor that
 * only had 8 bits per integer and 16 bits per long.
 * In that example, a 32 bit integer size is not even available.
 * This header file should be robust to that.
 *
 * For the case of an 8 bit processor, the preprocessor
 * may be limited to 16 bit math like its target.  That limitation
 * would mean that 32 bit comparisons can't be done accurately.
 * To increase robustness to this, comparisons are done against
 * smaller values first.  An inaccurate 32 bit comparison isn't
 * attempted if the 16 bit comparison has already succeeded.
 *
 * Limitations on preprocessor math can also be stricter than
 * for the target.  There are known cases where a compiler
 * targeting processors with 64 bit longs can't do accurate
 * preprocessor comparisons on more than 32 bits.
 */

/* Determine the number of bits for int, long, short, and char.
 * If one fails to be determined, set the number of bits to -1
 */

#ifndef TMW_BITS_PER_INT
# if   INT_MAX  == 0x7FL
#  define TMW_BITS_PER_INT 8
# elif INT_MAX  == 0x7FFFL
#  define TMW_BITS_PER_INT 16
# elif INT_MAX  == 0x7FFFFFFFL
#  define TMW_BITS_PER_INT 32
# else
#  define TMW_BITS_PER_INT -1
# endif
#endif

#ifndef TMW_BITS_PER_LONG
# if   LONG_MAX  == 0x7FL
#  define TMW_BITS_PER_LONG 8
# elif LONG_MAX  == 0x7FFFL
#  define TMW_BITS_PER_LONG 16
# elif LONG_MAX  == 0x7FFFFFFFL
#  define TMW_BITS_PER_LONG 32
# else
#  define TMW_BITS_PER_LONG -1
# endif
#endif

#ifndef TMW_BITS_PER_SHRT
# if   SHRT_MAX  == 0x7FL
#  define TMW_BITS_PER_SHRT 8
# elif SHRT_MAX  == 0x7FFFL
#  define TMW_BITS_PER_SHRT 16
# elif SHRT_MAX  == 0x7FFFFFFFL
#  define TMW_BITS_PER_SHRT 32
# else
#  define TMW_BITS_PER_SHRT -1
# endif
#endif

#ifndef TMW_BITS_PER_SCHAR
# if   SCHAR_MAX  == 0x7FL
#  define TMW_BITS_PER_SCHAR 8
# elif SCHAR_MAX  == 0x7FFFL
#  define TMW_BITS_PER_SCHAR 16
# elif SCHAR_MAX  == 0x7FFFFFFFL
#  define TMW_BITS_PER_SCHAR 32
# else
#  define TMW_BITS_PER_SCHAR -1
# endif
#endif

#ifndef TMW_CHAR_SIGNED
# if SCHAR_MAX == CHAR_MAX
#  define TMW_CHAR_SIGNED 1
# else
#  define TMW_CHAR_SIGNED 0
# endif
#endif

/* It is common for one or more of the integer types
 * to be the same size.  For example, on many embedded
 * processors, both shorts and ints are 16 bits.  On
 * processors used for workstations, it is quite common
 * for both int and long to be 32 bits.
 *   When there is more than one choice for typdef'ing
 * a portable type like int16_T or uint32_T, in
 * concept, it should not matter which choice is made.
 * However, some style guides and some code checking
 * tools do identify and complain about seemingly
 * irrelevant differences.  For example, a code
 * checking tool may complain about an implicit
 * conversion from int to short even though both
 * are 16 bits.  To reduce these types of
 * complaints, it is best to make int the
 * preferred choice when more than one is available.
 */

#ifndef INT8_T
# if   TMW_BITS_PER_INT   == 8
#  define  INT8_T int
# elif TMW_BITS_PER_LONG  == 8
#  define  INT8_T long
# elif TMW_BITS_PER_SCHAR == 8
#  define  INT8_T signed char
# elif TMW_BITS_PER_SHRT  == 8
#  define  INT8_T short
# endif
#endif
#ifdef INT8_T
 typedef INT8_T int8_T;
#endif

#ifndef UINT8_T
# if   TMW_BITS_PER_INT   == 8
#  define  UINT8_T unsigned int
# elif TMW_BITS_PER_LONG  == 8
#  define  UINT8_T unsigned long
# elif TMW_BITS_PER_SCHAR == 8
#  define  UINT8_T unsigned char
# elif TMW_BITS_PER_SHRT  == 8
#  define  UINT8_T unsigned short
# endif
#endif
#ifdef UINT8_T
 typedef UINT8_T uint8_T;
#endif

#ifndef INT16_T
# if   TMW_BITS_PER_INT   == 16
#  define  INT16_T int
# elif TMW_BITS_PER_LONG  == 16
#  define  INT16_T long
# elif TMW_BITS_PER_SCHAR == 16
#  define  INT16_T signed char
# elif TMW_BITS_PER_SHRT  == 16
#  define  INT16_T short
# endif
#endif
#ifdef INT16_T
 typedef INT16_T int16_T;
#endif

#ifndef UINT16_T
# if   TMW_BITS_PER_INT   == 16
#  define  UINT16_T unsigned int
# elif TMW_BITS_PER_LONG  == 16
#  define  UINT16_T unsigned long
# elif TMW_BITS_PER_SCHAR == 16
#  define  UINT16_T unsigned char
# elif TMW_BITS_PER_SHRT  == 16
#  define  UINT16_T unsigned short
# endif
#endif
#ifdef UINT16_T
 typedef UINT16_T uint16_T;
#endif

/* B&R specific define: */
# define INT32_T long

#ifndef INT32_T
# if   TMW_BITS_PER_INT   == 32
#  define  INT32_T int
# elif TMW_BITS_PER_LONG  == 32
#  define  INT32_T long
# elif TMW_BITS_PER_SCHAR == 32
#  define  INT32_T signed char
# elif TMW_BITS_PER_SHRT  == 32
#  define  INT32_T short
# endif
#endif
#ifdef INT32_T
 typedef INT32_T int32_T;
#endif

/* B&R specific define: */
# define UINT32_T unsigned long

#ifndef UINT32_T
# if   TMW_BITS_PER_INT   == 32
#  define  UINT32_T unsigned int
# elif TMW_BITS_PER_LONG  == 32
#  define  UINT32_T unsigned long
# elif TMW_BITS_PER_SCHAR == 32
#   define UINT32_T unsigned char
# elif TMW_BITS_PER_SHRT  == 32
#  define  UINT32_T unsigned short
# endif
#endif
#ifdef UINT32_T
 typedef UINT32_T uint32_T;
#endif

/* The following is used to emulate smaller integer types when only
 * larger types are available.  For example, compilers for TI C3x/C4x DSPs
 * define char and short to be 32 bits, so 8 and 16 bits are not directly
 * available.  This target is commonly used with RTW rapid prototyping.
 * Other DSPs define char to be 16 bits, so 8 bits is not directly
 * available.
 */
#ifndef INT8_T
# ifdef INT16_T
#  define INT8_T INT16_T
   typedef INT8_T int8_T;
# else
#  ifdef INT32_T
#   define INT8_T INT32_T
    typedef INT8_T int8_T;
#  endif
# endif
#endif

#ifndef UINT8_T
# ifdef UINT16_T
#   define UINT8_T UINT16_T
    typedef UINT8_T uint8_T;
# else
#  ifdef UINT32_T
#   define UINT8_T UINT32_T
    typedef UINT8_T uint8_T;
#  endif
# endif
#endif

#ifndef INT16_T
# ifdef INT32_T
#   define INT16_T INT32_T
    typedef INT16_T int16_T;
# endif
#endif

#ifndef UINT16_T
# ifdef UINT32_T
#   define UINT16_T UINT32_T
    typedef UINT16_T uint16_T;
# endif
#endif

#ifndef NO_FLOATS

#ifndef REAL32_T
# ifndef __MWERKS__
#  if FLT_MANT_DIG >= 23
#   define REAL32_T float
#  endif
# else
#  define REAL32_T float
# endif
#endif
#ifdef REAL32_T
 typedef REAL32_T real32_T;
#endif

#ifndef REAL64_T
# ifndef __MWERKS__
#  if DBL_MANT_DIG >= 52
#   define REAL64_T double
#  endif
# else
#  define REAL64_T double
# endif
#endif
#ifdef REAL64_T
 typedef REAL64_T real64_T;
#endif

#endif /* NO_FLOATS*/

/*=======================================================================*
 * Fixed width word size data types:                                     *
 *   int64_T                      - signed 64 bit integers               *
 *   uint64_T                     - unsigned 64 bit integers             *
 *=======================================================================*/

#ifndef INT64_T
# if defined(__APPLE__)
#  define INT64_T long long
#  define FMT64 "ll"
#  if defined(__LP64__) && !defined(INT_TYPE_64_IS_LONG)
#    define INT_TYPE_64_IS_LONG
#  endif
# elif (defined(__x86_64__) || defined(__LP64__))&& !defined(__MINGW64__)
#  define INT64_T long
#  define FMT64 "l"
#  if !defined(INT_TYPE_64_IS_LONG)
#    define INT_TYPE_64_IS_LONG
#  endif
# elif defined(_MSC_VER) || (defined(__BORLANDC__) && __BORLANDC__ >= 0x530) \
                         || (defined(__WATCOMC__)  && __WATCOMC__  >= 1100)
#  define INT64_T __int64
#  define FMT64 "I64"
# elif defined(__GNUC__) || defined(TMW_ENABLE_INT64) \
                         || defined(__LCC64__)
#  define INT64_T long long
#  define FMT64 "ll"
# endif
#endif

#if defined(INT64_T)
# if defined(__GNUC__) && \
    ((__GNUC__ > 2) || ((__GNUC__ == 2) && (__GNUC_MINOR__ >=9)))
  __extension__
# endif
 typedef INT64_T int64_T;
#endif

#ifndef UINT64_T
# if defined(__APPLE__)
#  define UINT64_T unsigned long long
#  define FMT64 "ll"
#  if defined(__LP64__) && !defined(INT_TYPE_64_IS_LONG)
#    define INT_TYPE_64_IS_LONG
#  endif
# elif (defined(__x86_64__) || defined(__LP64__))&& !defined(__MINGW64__)
#  define UINT64_T unsigned long
#  define FMT64 "l"
#  if !defined(INT_TYPE_64_IS_LONG)
#    define INT_TYPE_64_IS_LONG
#  endif
# elif defined(_MSC_VER) || (defined(__BORLANDC__) && __BORLANDC__ >= 0x530) \
                         || (defined(__WATCOMC__)  && __WATCOMC__  >= 1100)
#  define UINT64_T unsigned __int64
#  define FMT64 "I64"
# elif defined(__GNUC__) || defined(TMW_ENABLE_INT64) \
                         || defined(__LCC64__)
#  define UINT64_T unsigned long long
#  define FMT64 "ll"
# endif
#endif

#if defined(_WIN64) || (defined(__APPLE__) && defined(__LP64__)) \
                    || defined(__x86_64__) \
                    || defined(__LP64__)
#  define INT_TYPE_64_IS_SUPPORTED
#endif

#if defined(UINT64_T)
# if defined(__GNUC__) && \
    ((__GNUC__ > 2) || ((__GNUC__ == 2) && (__GNUC_MINOR__ >=9)))
  __extension__
# endif
 typedef UINT64_T uint64_T;
#endif

/*===========================================================================*
 * Format string modifiers for using size_t variables in printf statements.  *
 *===========================================================================*/

#ifndef FMT_SIZE_T
#  if (defined( __GNUC__ ) || defined(_STDC_C99))&& !defined(__MINGW64__)
#    define FMT_SIZE_T "z"
#  elif defined (__WATCOMC__)
#    define FMT_SIZE_T "l"
#  elif defined (_WIN32 )
#    define FMT_SIZE_T "I"
#  else
#    define FMT_SIZE_T "l"
#  endif
#endif

#ifndef FMT_PTRDIFF_T
#  if defined(__APPLE__)
#    define FMT_PTRDIFF_T "l"
#  elif defined( __GNUC__ ) || defined(_STDC_C99)
#    define FMT_PTRDIFF_T "t"
#  elif defined (__WATCOMC__)
#    define FMT_PTRDIFF_T "l"
#  elif defined (_WIN32 )
#    define FMT_PTRDIFF_T "I"
#  else
#    define FMT_PTRDIFF_T "l"
#  endif
#endif

/*===========================================================================*
 * General or logical data types where the word size is not guaranteed.      *
 *  real_T     - possible settings include real32_T or real64_T              *
 *  time_T     - possible settings include real32_T or real64_T              *
 *  boolean_T                                                                *
 *  char_T                                                                   *
 *  int_T                                                                    *
 *  uint_T                                                                   *
 *  byte_T                                                                   *
 *===========================================================================*/

#ifndef NO_FLOATS

#ifndef REAL_T
# ifdef REAL64_T
#  define REAL_T real64_T
# else
#  ifdef REAL32_T
#   define REAL_T real32_T
#  endif
# endif
#endif
#ifdef REAL_T
 typedef REAL_T real_T;
#endif

#ifndef TIME_T
# ifdef REAL_T
#  define TIME_T real_T
# endif
#endif
#ifdef TIME_T
 typedef TIME_T time_T;
#endif

#endif /* NO_FLOATS */

#ifndef BOOLEAN_T
# if defined(UINT8_T)
#  define BOOLEAN_T UINT8_T
# else
#  define BOOLEAN_T unsigned int
# endif
#endif
typedef BOOLEAN_T boolean_T;

#ifndef CHARACTER_T
# define CHARACTER_T char
#endif
typedef CHARACTER_T char_T;

#ifndef INTEGER_T
# define INTEGER_T long int
#endif
typedef INTEGER_T int_T;

#ifndef UINTEGER_T
# define UINTEGER_T unsigned
#endif
typedef UINTEGER_T uint_T;

#ifndef BYTE_T
# define BYTE_T unsigned char
#endif
typedef BYTE_T byte_T;

/*===========================================================================*
 * Define Complex Structures                                                 *
 *===========================================================================*/
#ifndef NO_FLOATS

#ifndef CREAL32_T
#  ifdef REAL32_T
    typedef struct {
      real32_T re, im;
    } creal32_T;
#    define CREAL32_T creal32_T
#  endif
#endif

#ifndef CREAL64_T
#  ifdef REAL64_T
    typedef struct {
      real64_T re, im;
    } creal64_T;
#    define CREAL64_T creal64_T
#  endif
#endif

#ifndef CREAL_T
#  ifdef REAL_T
    typedef struct {
      real_T re, im;
    } creal_T;
#    define CREAL_T creal_T
#  endif
#endif

#endif /* NO_FLOATS */

#ifndef CINT8_T
#  ifdef INT8_T
    typedef struct {
      int8_T re, im;
    } cint8_T;
#    define CINT8_T cint8_T
#  endif
#endif

#ifndef CUINT8_T
#  ifdef UINT8_T
    typedef struct {
      uint8_T re, im;
    } cuint8_T;
#    define CUINT8_T cuint8_T
#  endif
#endif

#ifndef CINT16_T
#  ifdef INT16_T
    typedef struct {
      int16_T re, im;
    } cint16_T;
#    define CINT16_T cint16_T
#  endif
#endif

#ifndef CUINT16_T
#  ifdef UINT16_T
    typedef struct {
      uint16_T re, im;
    } cuint16_T;
#    define CUINT16_T cuint16_T
#  endif
#endif

#ifndef CINT32_T
#  ifdef INT32_T
    typedef struct {
      int32_T re, im;
    } cint32_T;
#    define CINT32_T cint32_T
#  endif
#endif

#ifndef CUINT32_T
#  ifdef UINT32_T
    typedef struct {
      uint32_T re, im;
    } cuint32_T;
#    define CUINT32_T cuint32_T
#  endif
#endif

#ifndef CINT64_T
#  ifdef INT64_T
    typedef struct {
      int64_T re, im;
    } cint64_T;
#    define CINT64_T cint64_T
#  endif
#endif

#ifndef CUINT64_T
#  ifdef UINT64_T
    typedef struct {
      uint64_T re, im;
    } cuint64_T;
#    define CUINT64_T cuint64_T
#  endif
#endif

/*=======================================================================*
 * Min and Max:                                                          *
 *   int8_T, int16_T, int32_T     - signed 8, 16, or 32 bit integers     *
 *   uint8_T, uint16_T, uint32_T  - unsigned 8, 16, or 32 bit integers   *
 *=======================================================================*/

#define  MAX_int8_T      ((int8_T)(127))            /* 127  */
#define  MIN_int8_T      ((int8_T)(-128))           /* -128 */
#define  MAX_uint8_T     ((uint8_T)(255))           /* 255  */
#define  MIN_uint8_T     ((uint8_T)(0))

#define  MAX_int16_T     ((int16_T)(32767))         /* 32767 */
#define  MIN_int16_T     ((int16_T)(-32768))        /* -32768 */
#define  MAX_uint16_T    ((uint16_T)(65535))        /* 65535 */
#define  MIN_uint16_T    ((uint16_T)(0))

#define  MAX_int32_T     ((int32_T)(2147483647))    /* 2147483647  */
#define  MIN_int32_T     ((int32_T)(-2147483647-1)) /* -2147483648 */
#define  MAX_uint32_T    ((uint32_T)(0xFFFFFFFFU))  /* 4294967295  */
#define  MIN_uint32_T    ((uint32_T)(0))

#if defined(_MSC_VER) || (defined(__BORLANDC__) && __BORLANDC__ >= 0x530) \
                      || (defined(__WATCOMC__)  && __WATCOMC__  >= 1100) \
                      || defined(__LCC64__)
#  ifdef INT64_T
#    define  MAX_int64_T     ((int64_T)(9223372036854775807LL))
#    define  MIN_int64_T     ((int64_T)(-9223372036854775807LL-1LL))
#  endif
#  ifdef UINT64_T
#    define  MAX_uint64_T    ((uint64_T)(0xFFFFFFFFFFFFFFFFULL))
#    define  MIN_uint64_T    ((uint64_T)(0))
#  endif
#else
#  ifdef INT64_T
#    ifdef INT_TYPE_64_IS_LONG
#      define  MAX_int64_T     ((int64_T)(9223372036854775807L))
#      define  MIN_int64_T     ((int64_T)(-9223372036854775807L-1L))
#    else
#      define  MAX_int64_T     ((int64_T)(9223372036854775807LL))
#      define  MIN_int64_T     ((int64_T)(-9223372036854775807LL-1LL))
#    endif
#  endif
#  ifdef UINT64_T
#    ifdef INT_TYPE_64_IS_LONG
#      define  MAX_uint64_T    ((uint64_T)(0xFFFFFFFFFFFFFFFFUL))
#      define  MIN_uint64_T    ((uint64_T)(0))
#    else
#      define  MAX_uint64_T    ((uint64_T)(0xFFFFFFFFFFFFFFFFULL))
#      define  MIN_uint64_T    ((uint64_T)(0))
#    endif
#  endif
#endif

#ifdef _MSC_VER
/* Conversion from unsigned __int64 to double is not implemented in windows
 * and results in a compile error, thus the value must first be cast to
 * signed __int64, and then to double.
 *
 * If the 64 bit int value is greater than 2^63-1, which is the signed int64 max,
 * the macro below provides a workaround for casting a uint64 value to a double
 * in windows.
 */
#  define uint64_to_double(u) ( ((u) > _I64_MAX) ? \
            (double)(__int64)((u) - _I64_MAX - 1) + (double)_I64_MAX + 1: \
            (double)(__int64)(u) )

/* The following inline function should only be used in the macro double_to_uint64,
 * as it only handles the specfic range of double between 2^63 and 2^64-1 */
__forceinline
uint64_T double_to_uint64_helper(double d) {
  union double_to_uint64_union_type {
    double dd;
    uint64_T i64;
  } di;
  di.dd = d;
  return (((di.i64 & 0x000fffffffffffff) | 0x0010000000000000) << 11);
}

/* The largest double value that can be cast to uint64 in windows is the
 * signed int64 max, which is 2^63-1. The macro below provides
 * a workaround for casting large double values to uint64 in windows.
 */
/* The magic number 18446744073709551616.0 is 2^64 */
/* The magic number 9223372036854775808.0 is 2^63 */
#  define double_to_uint64(d) ( ((d) >= 18446744073709551616.0) ? \
            0xffffffffffffffffULL : \
            ((d) >= 0.0) ? \
            ((d) >= 9223372036854775808.0) ? \
            double_to_uint64_helper(d) : \
            (unsigned __int64)(d) : \
            0ULL )
#else
#  define uint64_to_double(u) ((double)(u))
#  if defined(__BORLANDC__) || defined(__WATCOMC__) || defined(__TICCSC__)
/* double_to_uint64 defined only for MSVC and UNIX */
#  else
#  define double_to_uint64(d) ( ((d) >= 18446744073709551616.0) ? \
            (unsigned long long) 0xffffffffffffffffULL : \
            ((d) >= 0) ? (unsigned long long)(d) : (unsigned long long) 0 )
#  endif
#endif

#if !defined(__cplusplus) && !defined(__bool_true_false_are_defined)

#ifndef _bool_T
#define _bool_T

typedef boolean_T bool;

#ifndef false
#define false (0)
#endif
#ifndef true
#define true (1)
#endif

#endif /* _bool_T */

#endif /* !__cplusplus */

/*
 * This software assumes that the code is being compiled on a target using a
 * 2's complement representation for signed integer values.
 */
#if ((SCHAR_MIN + 1) != -SCHAR_MAX)
#error "This code must be compiled using a 2's complement representation for signed integer values"
#endif

/*
 * Maximum length of a MATLAB identifier (function/variable/model)
 * including the null-termination character.
 */
#define TMW_NAME_LENGTH_MAX 64

/*
 * Maximum values for indices and dimensions
 */
#include <stddef.h>

#ifdef MX_COMPAT_32
typedef int mwSize;
typedef int mwIndex;
typedef int mwSignedIndex;
#else
typedef size_t    mwSize;         /* unsigned pointer-width integer */
typedef size_t    mwIndex;        /* unsigned pointer-width integer */
typedef ptrdiff_t mwSignedIndex;  /* a signed pointer-width integer */
#endif

#if (defined(_LP64) || defined(_WIN64)) && !defined(MX_COMPAT_32)
/* Currently 2^48 based on hardware limitations */
# define MWSIZE_MAX    281474976710655UL
# define MWINDEX_MAX   281474976710655UL
# define MWSINDEX_MAX  281474976710655L
# define MWSINDEX_MIN -281474976710655L
#else
# define MWSIZE_MAX    2147483647UL
# define MWINDEX_MAX   2147483647UL
# define MWSINDEX_MAX  2147483647L
# define MWSINDEX_MIN -2147483647L
#endif
#define MWSIZE_MIN    0UL
#define MWINDEX_MIN   0UL

/** UTF-16 character type */

#if (defined(__cplusplus) && (__cplusplus >= 201103L)) || (defined(_HAS_CHAR16_T_LANGUAGE_SUPPORT) && _HAS_CHAR16_T_LANGUAGE_SUPPORT)
typedef char16_t CHAR16_T;
#define U16_STRING_LITERAL_PREFIX u
#elif defined(_MSC_VER)
typedef wchar_t CHAR16_T;
#define U16_STRING_LITERAL_PREFIX L
#else
typedef UINT16_T CHAR16_T;
#endif

#endif  /* __TMWTYPES__ */

#endif /* tmwtypes_h */
```

### MessageServiceLayer.h
```c
/* Copyright 2013-2017 The MathWorks, Inc. */

#ifndef _message_service_layer_h_
#define _message_service_layer_h_

#ifdef SUPPORTS_PRAGMA_ONCE
#pragma once
#endif

#if defined(S_FUNCTION_NAME)
#include "mwmathutil.h"
#endif

typedef struct SimStruct_tag SimStruct;
typedef int int_T;

LIBMWSF_RUNTIME_API void* slMessageRtRegisterLocalMessageQueue(SimStruct* S, int queueId);
LIBMWSF_RUNTIME_API void* slMessageRtRegisterInputMessageQueue(SimStruct* S, int portNum);
LIBMWSF_RUNTIME_API void* slMessageRtRegisterOutputMessageQueue(SimStruct* S, int portNum);

LIBMWSF_RUNTIME_API void slMessageRtDiagnosticCheck(void* msgInterface, void* destMsgInterface, const char* diagnosticDesc, unsigned int ssid, int offsetSrcLoc, int lengthSrcLoc);
LIBMWSF_RUNTIME_API void slMessageRtSetQueueAttribute(void* msgInterface, const char* attribute, int value, const char* attribute2, int value2);

LIBMWSF_RUNTIME_API uint8_T slMessageRtHasOverflowOccurred(int status);
LIBMWSF_RUNTIME_API int slMessageRtMessageWasPopped(int status);
LIBMWSF_RUNTIME_API void slMessageRtDestroyQueue(void* msgInterface);

LIBMWSF_RUNTIME_API int slMessageRtSend(void* msgInterface, void* payload);
LIBMWSF_RUNTIME_API int slMessageRtReceive(void* msgInterface, void** payload);
LIBMWSF_RUNTIME_API int slMessageRtDesReceive(void* msgInterface, void** payload, bool isMsgTrigger);
LIBMWSF_RUNTIME_API int slMessageRtForward(void* msgInterfaceSrc, void* msgInterfaceDest);
LIBMWSF_RUNTIME_API void slMessageRtDestroyActiveMessageIfPresent(void* msgInterface);
LIBMWSF_RUNTIME_API int slMessageRtIsMessageValid(void* msgInterface);

LIBMWSF_RUNTIME_API int slMessageRtHasMessageBeenForwarded(void* msgInterface);

LIBMWSF_RUNTIME_API int_T slMessageRtLength(void* msgInterface);
LIBMWSF_RUNTIME_API void* slMessageRtPeek(void* msgInterface);
LIBMWSF_RUNTIME_API void* slMessageRtPeekAtIndex(void* msgInterface, int indexInQueue);

#endif
```

### sf_runtime_errors.h
```c
/* Copyright 2014-2017 The MathWorks, Inc. */

#ifndef RT_RUNTIME_ERRORS_H
#define RT_RUNTIME_ERRORS_H

#include "tmwtypes.h"
#include "sf_runtime/sf_runtime_spec.h"
#include "sf_runtime/utils.h"

struct SfDebugInstanceStruct;

typedef enum ThrowFlag
{
    ThrowFlag_MESSAGE = -4,
    ThrowFlag_WARNING = -2,
    ThrowFlag_NONE = -1,
    ThrowFlag_SAFE_ERROR = 0,
    ThrowFlag_ERROR = 1,
} ThrowFlag;

LIBMWSF_RUNTIME_API void sf_read_before_write_error(SimStruct* S,
                                                    unsigned int dataNumber,
                                                    unsigned int ssIdOfSourceObject,
                                                    int offsetInSourceObject,
                                                    int lengthInSourceObject);

LIBMWSF_RUNTIME_API double sf_data_range_check_min_max(SimStruct* S,
                                                       unsigned int ssIdOfSourceObject,
                                                       int offsetInSourceObject,
                                                       int lengthInSourceObject,
                                                       unsigned int dataNumber,
                                                       double dataValue,
                                                       double dataMin,
                                                       double dataMax);

LIBMWSF_RUNTIME_API double sf_data_range_check_max(SimStruct* S,
                                                   unsigned int ssIdOfSourceObject,
                                                   int offsetInSourceObject,
                                                   int lengthInSourceObject,
                                                   unsigned int dataNumber,
                                                   double dataValue,
                                                   double dataMax);

LIBMWSF_RUNTIME_API double sf_data_range_check_min(SimStruct* S,
                                                   unsigned int ssIdOfSourceObject,
                                                   int offsetInSourceObject,
                                                   int lengthInSourceObject,
                                                   unsigned int dataNumber,
                                                   double dataValue,
                                                   double dataMin);

LIBMWSF_RUNTIME_API void sf_state_inconsistency_error(SimStruct* S,
                                                      unsigned int ssIdOfSourceObject);

LIBMWSF_RUNTIME_API void sf_cycle_depth_limit_error(SimStruct* S,
                                                    unsigned int ssIdOfSourceObject, unsigned int recursionLimit);

LIBMWSF_RUNTIME_API int sf_array_bounds_check(struct SfDebugInstanceStruct* debugInstance,
                                              SimStruct* S,
                                              unsigned int ssIdOfSourceObject,
                                              int offsetInSourceObject,
                                              int lengthInSourceObject,
                                              int dataNumber,
                                              int indexValue,
                                              int firstIndex,
                                              int lastIndex);

LIBMWSF_RUNTIME_API int sf_eml_array_bounds_check(struct SfDebugInstanceStruct* debugInstance,
                                                  SimStruct* S,
                                                  unsigned int ssIdOfSourceObject,
                                                  int offsetInSourceObject,
                                                  int lengthInSourceObject,
                                                  int dataNumber,
                                                  int indexValue,
                                                  int firstIndex,
                                                  int lastIndex);

#ifdef INT_TYPE_64_IS_SUPPORTED
LIBMWSF_RUNTIME_API int64_T sf_eml_array_bounds_check_int64(struct SfDebugInstanceStruct* debugInstance,
                                                            SimStruct* S,
                                                            unsigned int ssIdOfSourceObject,
                                                            int offsetInSourceObject,
                                                            int lengthInSourceObject,
                                                            int dataNumber,
                                                            int64_T indexValue,
                                                            int64_T firstIndex,
                                                            int64_T lastIndex);
#endif

LIBMWSF_RUNTIME_API int sf_eml_shift_index_bounds_check(struct SfDebugInstanceStruct* debugInstance,
                                                        SimStruct* S,
                                                        unsigned int ssIdOfSourceObject,
                                                        int offsetInSourceObject,
                                                        int lengthInSourceObject,
                                                        const char* operandText,
                                                        int indexValue,
                                                        int firstIndex,
                                                        int lastIndex);

#ifdef INT_TYPE_64_IS_SUPPORTED
LIBMWSF_RUNTIME_API int64_T sf_eml_shift_index_bounds_check_int64(struct SfDebugInstanceStruct* debugInstance,
                                                                  SimStruct* S,
                                                                  unsigned int ssIdOfSourceObject,
                                                                  int offsetInSourceObject,
                                                                  int lengthInSourceObject,
                                                                  const char* operandText,
                                                                  int64_T indexValue,
                                                                  int64_T firstIndex,
                                                                  int64_T lastIndex);
#endif

LIBMWSF_RUNTIME_API int sf_type_range_check(struct SfDebugInstanceStruct* debugInstance,
                                            SimStruct* S,
                                            unsigned int ssIdOfSourceObject,
                                            int offsetInSourceObject,
                                            int lengthInSourceObject,
                                            int indexValue,
                                            int firstIndex,
                                            int lastIndex);

LIBMWSF_RUNTIME_API int sf_eml_type_range_check(struct SfDebugInstanceStruct* debugInstance,
                                                SimStruct* S,
                                                unsigned int ssIdOfSourceObject,
                                                int offsetInSourceObject,
                                                int lengthInSourceObject,
                                                int indexValue,
                                                int firstValue,
                                                int lastIndex);

#ifdef INT_TYPE_64_IS_SUPPORTED
LIBMWSF_RUNTIME_API int64_T sf_eml_type_range_check_int64(struct SfDebugInstanceStruct* debugInstance,
                                                          SimStruct* S,
                                                          unsigned int ssIdOfSourceObject,
                                                          int offsetInSourceObject,
                                                          int lengthInSourceObject,
                                                          int64_T indexValue,
                                                          int64_T firstIndex,
                                                          int64_T lastIndex);

#endif

LIBMWSF_RUNTIME_API void sf_array_size_mismatch_error(SimStruct* S, unsigned int ssIdOfSourceObject, int offsetInSourceObject, int lengthInSourceObject,
                                                      unsigned int dimension, const char* arrayName1, int size1, const char* arrayName2, int size2);
LIBMWSF_RUNTIME_API void sf_data_overflow_error(SimStruct* S, unsigned int ssIdOfSourceObject, int offsetInSourceObject, int lengthInSourceObject);

LIBMWSF_RUNTIME_API void sf_data_saturate_error(SimStruct* S, unsigned int ssIdOfSourceObject, int offsetInSourceObject, int lengthInSourceObject);
LIBMWSF_RUNTIME_API void sf_data_divide_by_zero_error(SimStruct* S, unsigned int ssIdOfSourceObject, int offsetInSourceObject, int lengthInSourceObject);
LIBMWSF_RUNTIME_API void sf_data_range_error(SimStruct* S, unsigned int ssIdOfSourceObject, int offsetInSourceObject, int lengthInSourceObject, unsigned int dataNumber, double dataValue, double* dataMin, double* dataMax);
LIBMWSF_RUNTIME_API double sf_integer_check(SimStruct* S, unsigned int ssIdOfSourceObject, int offsetInSourceObject, int lengthInSourceObject, double value);
LIBMWSF_RUNTIME_API void sf_unsafe_enum_cast_error(SimStruct* S, unsigned int ssIdOfSourceObject, int offsetInSourceObject, int lengthInSourceObject);

LIBMWSF_RUNTIME_API void sf_attempt_to_access_forwarded_message_error(SimStruct* S, unsigned int ssIdOfSourceObject, int offsetInSourceObject, int lengthInSourceObject);
LIBMWSF_RUNTIME_API void sf_attempt_to_discard_unavailable_message_error(SimStruct* S, unsigned int ssIdOfSourceObject, int offsetInSourceObject, int lengthInSourceObject);
LIBMWSF_RUNTIME_API void sf_attempt_to_forward_unpopped_message_error(SimStruct* S, unsigned int ssIdOfSourceObject, int offsetInSourceObject, int lengthInSourceObject);
LIBMWSF_RUNTIME_API void sf_attempt_to_update_payload_before_pop_error(SimStruct* S, unsigned int ssIdOfSourceObject, int offsetInSourceObject, int lengthInSourceObject);
LIBMWSF_RUNTIME_API void sf_attempt_to_update_payload_for_forwarded_message_error(SimStruct* S, unsigned int ssIdOfSourceObject, int offsetInSourceObject, int lengthInSourceObject);
LIBMWSF_RUNTIME_API void sf_attempt_to_read_payload_before_pop_error(SimStruct* S, unsigned int ssIdOfSourceObject, int offsetInSourceObject, int lengthInSourceObject);
LIBMWSF_RUNTIME_API void sf_attempt_to_read_payload_for_forwarded_message_error(SimStruct* S, unsigned int ssIdOfSourceObject, int offsetInSourceObject, int lengthInSourceObject);
LIBMWSF_RUNTIME_API void sf_attempt_to_read_queue_overflow_var_before_pop_error(SimStruct* S, unsigned int ssIdOfSourceObject, int offsetInSourceObject, int lengthInSourceObject);
LIBMWSF_RUNTIME_API void sf_msg_queue_overflow_error(SimStruct* S, unsigned int ssIdOfSourceObject, int offsetInSourceObject, int lengthInSourceObject);
LIBMWSF_RUNTIME_API void sf_msg_queue_overflow_warning(SimStruct* S, unsigned int ssIdOfSourceObject, int offsetInSourceObject, int lengthInSourceObject);
LIBMWSF_RUNTIME_API void sf_msg_overflow_information_for_local_queue(SimStruct* S, const char* queueName, int numDroppedMessages, int recommendedQueueCapacity);

LIBMWSF_RUNTIME_API ThrowFlag getSimulinkParameterMode(SimStruct* S, const char *modelName, const char *parameter);

void sf_stop_simulation();

#endif
```
